// TIA Portal V17 export
// export: Created 2022-10-14T12:26:42.7495408Z, ExportSetting WithDefaults, DisplayName Totally Integrated Automation Portal, DisplayVersion V17 Update 4, DisplayName TIA Portal Openness, DisplayVersion V17 Update 4, DisplayName TIA Portal Version Control Interface, DisplayVersion V17, DisplayName SINAMICS Startdrive Advanced, DisplayVersion V17 Update2, DisplayName SINAMICS Startdrive G130, G150, S120, S150, SINAMICS MV, S210, DisplayVersion V17 Update2, DisplayName SINAMICS Startdrive G110M, G120, G120C, G120D, G120P, G115D, DisplayVersion V17 Update2, DisplayName STEP 7 Professional, DisplayVersion V17 Update 4, DisplayName STEP 7 Safety, DisplayVersion V17, DisplayName WinCC Advanced / Unified PC, DisplayVersion V17 Update 4
FUNCTION "1000_IT_Aufruf" : Void   // FC1000, FBD
TITLE = Haupt aufruf
{ S7_Optimized_Access := 'TRUE' }
VERSION : 0.1
// stored: AutoNumber false, IsIECCheckEnabled false, SetENOAutomatically false, UDAEnableTagReadback false
BEGIN

REGION Network 1
   // Bender-gerät kommunikation baustein (COM465ID)
   //                               FEST GmbH  
   //  M.Alsouki            27.11.2019     v 1.04
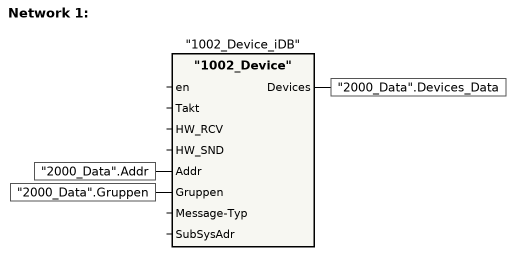
   "1002_Device_iDB"(Addr := "2000_Data".Addr,   // "1002_Device"
                     Gruppen := "2000_Data".Gruppen,
                     Devices => "2000_Data".Devices_Data);
END_REGION
END_FUNCTION
